// Mitsubishi GX Works2 project: 2023-06-07 #2 생산자동화기능사 12번   PLC: Q03UDV
// 생산자동화기능사

// global labels: Global1
VAR_GLOBAL
  PB1 AT X0 : BOOL;
  PB2 AT X1 : BOOL;
  정지 AT X2 : BOOL;
  공급후진 AT X3 : BOOL;
  공급전진 AT X4 : BOOL;
  가공후진 AT X5 : BOOL;
  가공전진 AT X6 : BOOL;
  송출후진 AT X7 : BOOL;
  송출전진 AT X8 : BOOL;
  배출후진 AT X9 : BOOL;
  배출전진 AT X0A : BOOL;
  매거진 AT X0B : BOOL;
  금속센서 AT X0F : BOOL;
  PB3 AT X0C : BOOL;
  적 AT Y20 : BOOL;
  황 AT Y21 : BOOL;
  녹 AT Y22 : BOOL;
  공급1 AT Y23 : BOOL;
  공급2 AT Y24 : BOOL;
  가공 AT Y25 : BOOL;
  드릴 AT Y26 : BOOL;
  송출 AT Y27 : BOOL;
  배출 AT Y28 : BOOL;
  컨베이어 AT Y29 : BOOL;
END_VAR

PROGRAM 테스트동작
VAR
  PHASE : INT;
END_VAR
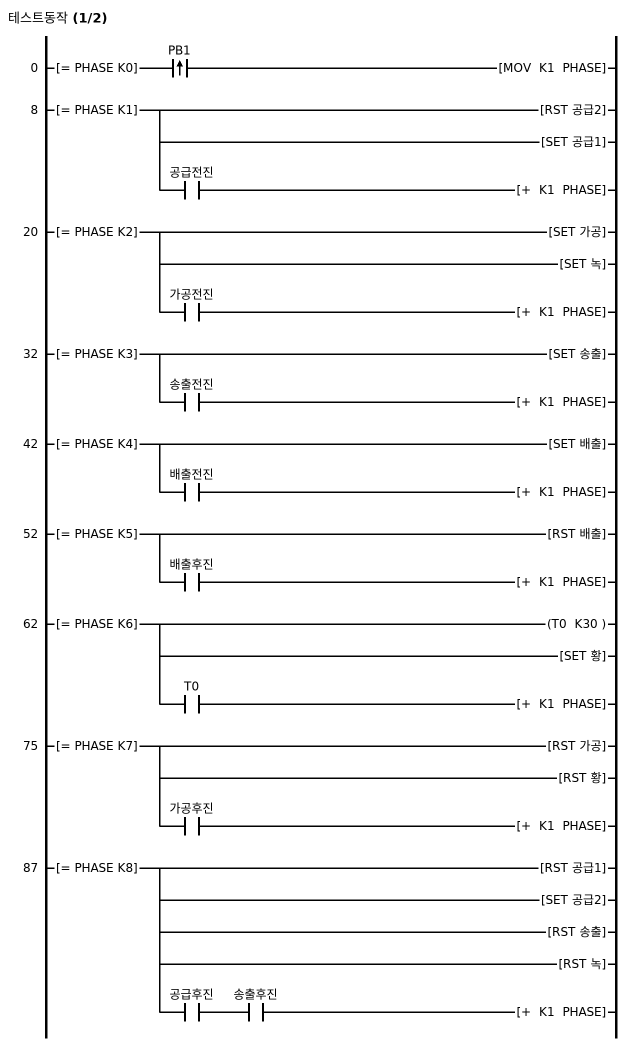
0     LD=     PHASE K0
      ANDP    PB1
      MOV     K1 PHASE
8     LD=     PHASE K1
      RST     공급2
      SET     공급1
      AND     공급전진
      +       K1 PHASE
20    LD=     PHASE K2
      SET     가공
      SET     녹
      AND     가공전진
      +       K1 PHASE
32    LD=     PHASE K3
      SET     송출
      AND     송출전진
      +       K1 PHASE
42    LD=     PHASE K4
      SET     배출
      AND     배출전진
      +       K1 PHASE
52    LD=     PHASE K5
      RST     배출
      AND     배출후진
      +       K1 PHASE
62    LD=     PHASE K6
      OUT     T0 K30
      SET     황
      AND     T0
      +       K1 PHASE
75    LD=     PHASE K7
      RST     가공
      RST     황
      AND     가공후진
      +       K1 PHASE
87    LD=     PHASE K8
      RST     공급1
      SET     공급2
      RST     송출
      RST     녹
      AND     공급후진
      AND     송출후진
      +       K1 PHASE
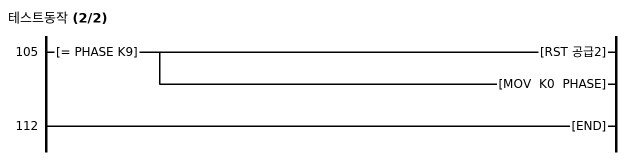
105   LD=     PHASE K9
      RST     공급2
      MOV     K0 PHASE
112   END
END_PROGRAM

PROGRAM 생산자동화기능사
VAR
  PHASE : INT;
  MODE : INT;
END_VAR
VAR CONSTANT
  단속 : INT;
  연속 : INT := 1;
END_VAR
VAR
  METAL : INT;
END_VAR
VAR CONSTANT
  금속 : INT := 1;
  비금속 : INT := 2;
END_VAR
VAR
  CNT1 : INT;
  CNT2 : INT;
  BLINK1 : ARRAY [0..3] OF BOOL;
  BLINK2 : ARRAY [0..3] OF BOOL;
  EMG : INT;
  BLINK3 : ARRAY [0..3] OF BOOL;
END_VAR
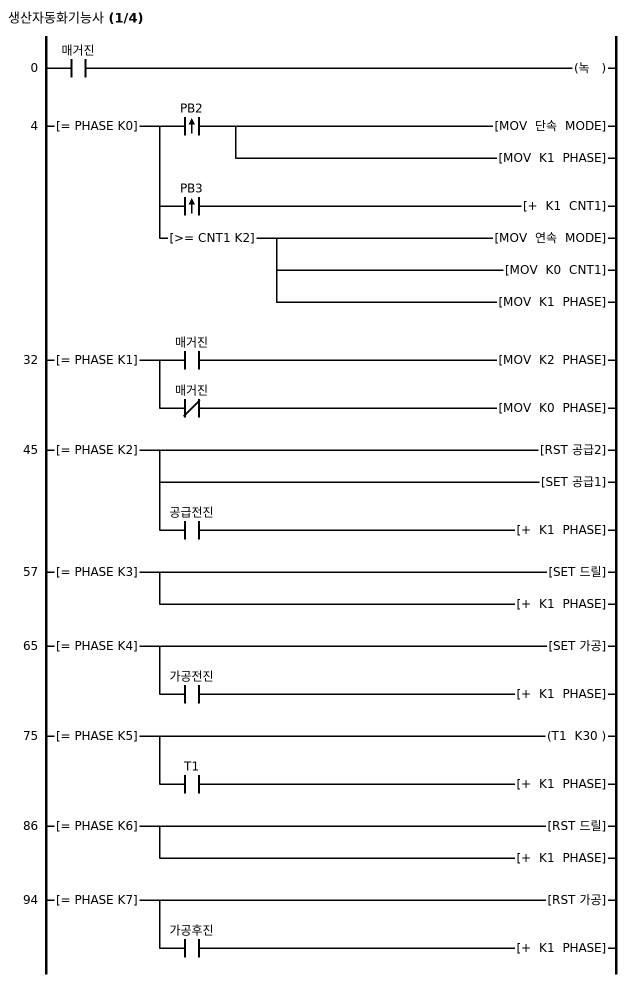
0     LD      매거진
      OUT     녹
4     LD=     PHASE K0
      MPS
      ANDP    PB2
      MOV     단속 MODE
      MOV     K1 PHASE
      MRD
      ANDP    PB3
      +       K1 CNT1
      MPP
      AND>=   CNT1 K2
      MOV     연속 MODE
      MOV     K0 CNT1
      MOV     K1 PHASE
32    LD=     PHASE K1
      MPS
      AND     매거진
      MOV     K2 PHASE
      MPP
      ANI     매거진
      MOV     K0 PHASE
45    LD=     PHASE K2
      RST     공급2
      SET     공급1
      AND     공급전진
      +       K1 PHASE
57    LD=     PHASE K3
      SET     드릴
      +       K1 PHASE
65    LD=     PHASE K4
      SET     가공
      AND     가공전진
      +       K1 PHASE
75    LD=     PHASE K5
      OUT     T1 K30
      AND     T1
      +       K1 PHASE
86    LD=     PHASE K6
      RST     드릴
      +       K1 PHASE
94    LD=     PHASE K7
      RST     가공
      AND     가공후진
      +       K1 PHASE
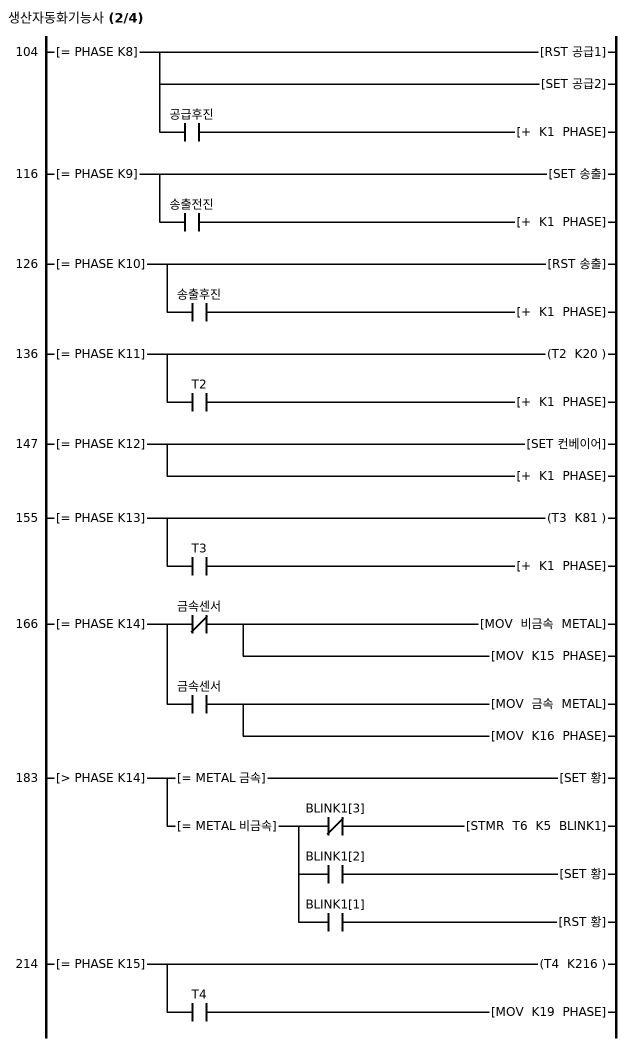
104   LD=     PHASE K8
      RST     공급1
      SET     공급2
      AND     공급후진
      +       K1 PHASE
116   LD=     PHASE K9
      SET     송출
      AND     송출전진
      +       K1 PHASE
126   LD=     PHASE K10
      RST     송출
      AND     송출후진
      +       K1 PHASE
136   LD=     PHASE K11
      OUT     T2 K20
      AND     T2
      +       K1 PHASE
147   LD=     PHASE K12
      SET     컨베이어
      +       K1 PHASE
155   LD=     PHASE K13
      OUT     T3 K81
      AND     T3
      +       K1 PHASE
166   LD=     PHASE K14
      MPS
      ANI     금속센서
      MOV     비금속 METAL
      MOV     K15 PHASE
      MPP
      AND     금속센서
      MOV     금속 METAL
      MOV     K16 PHASE
183   LD>     PHASE K14
      MPS
      AND=    METAL 금속
      SET     황
      MPP
      AND=    METAL 비금속
      MPS
      ANI     BLINK1[3]
      STMR    T6 K5 BLINK1
      MRD
      AND     BLINK1[2]
      SET     황
      MPP
      AND     BLINK1[1]
      RST     황
214   LD=     PHASE K15
      OUT     T4 K216
      AND     T4
      MOV     K19 PHASE
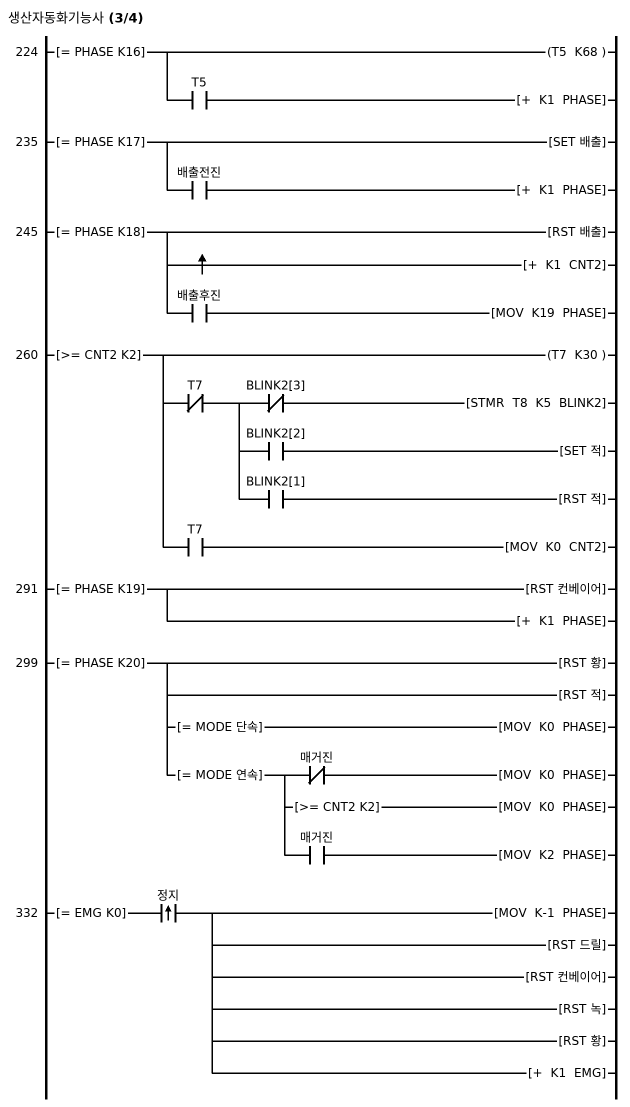
224   LD=     PHASE K16
      OUT     T5 K68
      AND     T5
      +       K1 PHASE
235   LD=     PHASE K17
      SET     배출
      AND     배출전진
      +       K1 PHASE
245   LD=     PHASE K18
      RST     배출
      MPS
      MEP
      +       K1 CNT2
      MPP
      AND     배출후진
      MOV     K19 PHASE
260   LD>=    CNT2 K2
      OUT     T7 K30
      MPS
      ANI     T7
      MPS
      ANI     BLINK2[3]
      STMR    T8 K5 BLINK2
      MRD
      AND     BLINK2[2]
      SET     적
      MPP
      AND     BLINK2[1]
      RST     적
      MPP
      AND     T7
      MOV     K0 CNT2
291   LD=     PHASE K19
      RST     컨베이어
      +       K1 PHASE
299   LD=     PHASE K20
      RST     황
      RST     적
      MPS
      AND=    MODE 단속
      MOV     K0 PHASE
      MPP
      AND=    MODE 연속
      MPS
      ANI     매거진
      MOV     K0 PHASE
      MRD
      AND>=   CNT2 K2
      MOV     K0 PHASE
      MPP
      AND     매거진
      MOV     K2 PHASE
332   LD=     EMG K0
      ANDP    정지
      MOV     K-1 PHASE
      RST     드릴
      RST     컨베이어
      RST     녹
      RST     황
      +       K1 EMG
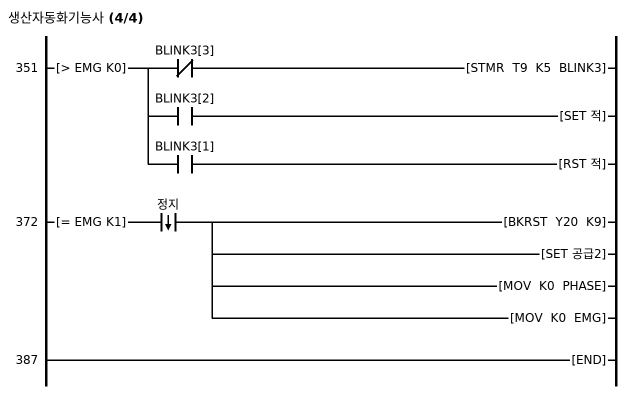
351   LD>     EMG K0
      MPS
      ANI     BLINK3[3]
      STMR    T9 K5 BLINK3
      MRD
      AND     BLINK3[2]
      SET     적
      MPP
      AND     BLINK3[1]
      RST     적
372   LD=     EMG K1
      ANDF    정지
      BKRST   Y20 K9
      SET     공급2
      MOV     K0 PHASE
      MOV     K0 EMG
387   END
END_PROGRAM
